(* CODESYS project CtaVisApps_1.0.0.0.library
   DocFormat: reStructuredText
   DefaultNamespace: CtaVisApps
   Version: 1.0.0.0
   Placeholder: CtaVisApps
   Company: CTA
   Description: Visu Apps Library der CTA
   CompiledLibraryCompatibilityVersion: CODESYS V3.5 SP16 Patch 3
   LanguageModelAttribute: qualified-access-only
   Title: CtaVisApps
   Author: SIS

Project tree, tasks and I/O mapping:
  libraries: CmpBitmapPool, 3.5.17.0 (System); Visu Utils, 4.5.0.0 (System); Standard, 3.5.18.0 (System); VisuElemBase, * (System); CtaVisSymbols, 1.0.0.0 (CTA); TextListUtils, * (System); VisuSymbols, 4.5.0.0 (System)
  40 Visualizations/
    APP/
      visualisation VIS_APP_BASE
      visualisation VIS_APP
    DESCTOP/
      visualisation VIS_DESCTOP_GVL
      visualisation VIS_DESCTOP_BASE
      visualisation VIS_DESCTOP_APP_LINE
      visualisation VIS_DESCTOP
  30 Program Organization Units/
    APP/
      function block FB_APP [ST]: DIALOG_NAME, ITF_BIG_SYBIL, ITF_LOW_SYBIL, ITF_PARENT, TEXTLIST, TEXTLISTID, PRESS_EVENT, ITF_CHILD, FB_INIT, ITF_SELF, ENABLED, DATA, DATA_SIZE, RELOAD_REQUEST, APP_NAME, ITF_DESCTOP
    DESCTOP/
      function block FB_DESCTOP [ST]: GET_APP, FIRST_APP, RETURN_APP, PATH, DialogClosed, LOWEST_CHILD, HOME, RELOAD_REQUEST
  00000000-0000-0000-0000-000000000000|D:\CoDeSys\LibrariesV3\trunk\Intern\CAA\CAA Template\3.4.0.0 draft\Placeholder.xml
  00000000-0000-0000-0000-000000000000|D:\CoDeSys\LibrariesV3\trunk\Intern\CAA\CAA Template\3.2.0.3 draft\Prefix.pdf
  00000000-0000-0000-0000-000000000000|D:\CoDeSys\LibrariesV3\trunk\Intern\CAA\CAA Template\3.5.2.0 draft\Placeholder.xml
  20 Structs/
  50 Images/
  10 Documenation/
    global variables VersionHistory
    global variables readMe
  21 Interface/
    interface ITF_APP: DIALOG_NAME, ITF_BIG_SYBIL, TEXTLISTID, ITF_LOW_SYBIL, TEXTLIST, PRESS_EVENT, ITF_CHILD, ITF_PARENT, ITF_SELF, ENABLED, DATA, DATA_SIZE, RELOAD_REQUEST, APP_NAME, ITF_DESCTOP
    interface ITF_DESCTOP: FIRST_APP, GET_APP, RETURN_APP, PATH, LOWEST_CHILD, HOME, RELOAD_REQUEST
  11 Library Parameter/
  12 Konstanten/
  60 Textlisten/
  13 Globale Variablen/
    global variables GVL_VISU_APPS
  5ce3da45-db07-42e7-a21c-a00fff4ed8f6|Icons\alert.svg
  5ce3da45-db07-42e7-a21c-a00fff4ed8f6|Icons\arrow-down.svg
  5ce3da45-db07-42e7-a21c-a00fff4ed8f6|Icons\arrow-down_square.svg
  5ce3da45-db07-42e7-a21c-a00fff4ed8f6|Icons\arrow-left_solo_black.svg
  5ce3da45-db07-42e7-a21c-a00fff4ed8f6|Icons\arrow-right_solo_black.svg
  5ce3da45-db07-42e7-a21c-a00fff4ed8f6|Icons\arrow-up.svg
  5ce3da45-db07-42e7-a21c-a00fff4ed8f6|Icons\calendar-range.svg
  5ce3da45-db07-42e7-a21c-a00fff4ed8f6|Icons\check.svg
  5ce3da45-db07-42e7-a21c-a00fff4ed8f6|Icons\clock-outline.svg
  5ce3da45-db07-42e7-a21c-a00fff4ed8f6|Icons\close_solo_black.svg
  5ce3da45-db07-42e7-a21c-a00fff4ed8f6|Icons\CtaInfo.svg
  5ce3da45-db07-42e7-a21c-a00fff4ed8f6|Icons\database_black.svg
  5ce3da45-db07-42e7-a21c-a00fff4ed8f6|Icons\delete_solo_black.svg
  5ce3da45-db07-42e7-a21c-a00fff4ed8f6|Icons\engine.svg
  5ce3da45-db07-42e7-a21c-a00fff4ed8f6|Icons\front_hand_Black.svg
  5ce3da45-db07-42e7-a21c-a00fff4ed8f6|Icons\front_hand_Yellow_Off.svg
  5ce3da45-db07-42e7-a21c-a00fff4ed8f6|Icons\gear.svg
  5ce3da45-db07-42e7-a21c-a00fff4ed8f6|Icons\home.svg
  5ce3da45-db07-42e7-a21c-a00fff4ed8f6|Icons\information-variant.svg
  5ce3da45-db07-42e7-a21c-a00fff4ed8f6|Icons\lightning-bolt-circle.svg
  5ce3da45-db07-42e7-a21c-a00fff4ed8f6|Icons\message.svg
  5ce3da45-db07-42e7-a21c-a00fff4ed8f6|Icons\message-alert-variant.svg
  5ce3da45-db07-42e7-a21c-a00fff4ed8f6|Icons\minus_solo_black.svg
  5ce3da45-db07-42e7-a21c-a00fff4ed8f6|Icons\plus_solo_black.svg
  5ce3da45-db07-42e7-a21c-a00fff4ed8f6|Icons\power_solo_black.svg
  5ce3da45-db07-42e7-a21c-a00fff4ed8f6|Icons\refresh_solo_black.svg
  5ce3da45-db07-42e7-a21c-a00fff4ed8f6|Icons\SearchFilter.svg
  5ce3da45-db07-42e7-a21c-a00fff4ed8f6|Icons\signal-celular-alt.svg
  5ce3da45-db07-42e7-a21c-a00fff4ed8f6|Icons\toggle-switch.svg
  5ce3da45-db07-42e7-a21c-a00fff4ed8f6|Icons\Modbus_Organization_Logo.svg
  5ce3da45-db07-42e7-a21c-a00fff4ed8f6|Icons\CheckboxUnchecked_withe.svg
  5ce3da45-db07-42e7-a21c-a00fff4ed8f6|Icons\lock_open_black.svg
  5ce3da45-db07-42e7-a21c-a00fff4ed8f6|Icons\check_green.svg
  5ce3da45-db07-42e7-a21c-a00fff4ed8f6|Icons\filter_black.svg
  5ce3da45-db07-42e7-a21c-a00fff4ed8f6|Icons\CtaLogo.png
  5ce3da45-db07-42e7-a21c-a00fff4ed8f6|Icons\Grafana_Logo.svg
  5ce3da45-db07-42e7-a21c-a00fff4ed8f6|Icons\hourglass_top.svg
  text list GlobalTextList
*)

// 10 Documenation/VersionHistory
(* 

.. image:: ../../Images/CTA_Logo.jpg
   :align: right
   :width: 15% 

**History**   


============ =========== =========== ============================================
**Date**     **Version** **Author**  **Change**
------------ ----------- ----------- --------------------------------------------
04.09.2023   0.0.0.1     SIS         Entwicklung Apps

============ =========== =========== ============================================


*)
VAR_GLOBAL
    stInfo : STRING:= '0.0.0.0, Vorlage, CTA';
END_VAR

// 10 Documenation/readMe
(*

**ReadMe**
 
|	**Empfehlung**
|
|	Mithilfe der CtaVisApps Library kann ein App Desctop erstellt werden mit minimalem Aufwand. Dazu muss die Visualisierung VIS_DESCTOP im Projekt implementiert werden.
|     
| *Beispiel*
+-----------------------+---------------------------------------------------------------------------------------------------------------------------------------------------------------------------------------------------------------------------------------------------------------------------------------------------------------------------------------------------------------------------------------------------------------------------------------+
| Beschreibung          |  Code                                                                                                                                                                                                                                                                                                                                                                                                                                 |
+=======================+=======================================================================================================================================================================================================================================================================================================================================================================================================================================+
| Deklaration           | .. code-block:: codesys                                                                                                                                                                                                                                                                                                                                                                                                               |
|                       |                                                                                                                                                                                                                                                            																																											|
|                       | 		APP_PFC200									:	CtaVisApps.FB_APP(0				,0)					:= 			(_ENABLED := TRUE,    _TEXTLIST	:= 'APPS',		_TEXTLISTID		:= 'PFC200',		_DIALOG_NAME	:= 'DIA_WBM');                       																																							            |
|                       |		APP_Management								:	CtaVisApps.FB_APP(0				,APP_PFC200)		:= 			(_ENABLED := TRUE,    _TEXTLIST	:= 'APPS',		_TEXTLISTID		:= 'MANAGEMENT',	_DIALOG_NAME	:= 'DIA_AnlagenManagement');     																																										 	|
|                       |   	APP_STVDA									: 	CtaVisApps.FB_APP(0				,APP_Management)	:= 			(_ENABLED := TRUE,    _TEXTLIST	:= 'APPS',		_TEXTLISTID		:= 'STVDA',			_DIALOG_NAME	:= ''	);                       																																									      	|
|						|			APP_F100								:	CtaVisApps.FB_APP(APP_STVDA		,0)					:= 			(_ENABLED := TRUE,    _TEXTLIST	:= 'APPS',		_TEXTLISTID		:= 'F100',			_DIALOG_NAME	:= ''	);                       																																							            	|
|						|				APP_F100S1							:	CtaVisApps.FB_APP(APP_F100		,0)					:= 			(_ENABLED := TRUE,    _TEXTLIST	:= 'APPS',		_TEXTLISTID		:= 'F100S1',		_DIALOG_NAME	:= ''	);                       																																									      	|
|                       | 					APP_100B011						:	CtaVisApps.FB_APP(APP_F100S1	,0)					:= 			(_ENABLED := TRUE,    _TEXTLIST	:= 'APPS',		_TEXTLISTID		:= '100B011',		_DIALOG_NAME	:= ''	);                       																																										 	|
| 						|					APP_100B012						:	CtaVisApps.FB_APP(APP_F100S1	,APP_100B011)		:= 			(_ENABLED := TRUE,    _TEXTLIST	:= 'APPS',		_TEXTLISTID		:= '100B012',		_DIALOG_NAME	:= ''	);                       																																											|
| 						|				APP_F100S2							:	CtaVisApps.FB_APP(APP_F100		,APP_F100S1)		:= 			(_ENABLED := TRUE,    _TEXTLIST	:= 'APPS',		_TEXTLISTID		:= 'F100S2',		_DIALOG_NAME	:= ''	);                       																																											|
| 						|					APP_100M021						:	CtaVisApps.FB_APP(APP_F100S2	,0)					:= 			(_ENABLED := TRUE,    _TEXTLIST	:= 'APPS',		_TEXTLISTID		:= '100M021',		_DIALOG_NAME	:= ''	);                       																																											|
| 						|				APP_F100S3							:	CtaVisApps.FB_APP(APP_F100		,APP_F100S2)		:= 			(_ENABLED := TRUE,    _TEXTLIST	:= 'APPS',		_TEXTLISTID		:= 'F100S3',		_DIALOG_NAME	:= ''	);                       																																											|
| 						|					APP_100M031						:	CtaVisApps.FB_APP(APP_F100S3	,0)					:= 			(_ENABLED := TRUE,    _TEXTLIST	:= 'APPS',		_TEXTLISTID		:= '100M031',		_DIALOG_NAME	:= ''	);                       																																											|
| 						|					APP_100M032						:	CtaVisApps.FB_APP(APP_F100S3	,APP_100M031)		:= 			(_ENABLED := TRUE,    _TEXTLIST	:= 'APPS',		_TEXTLISTID		:= '100M032',		_DIALOG_NAME	:= ''	);                       																																											|
| 						| 				APP_F100S4							:	CtaVisApps.FB_APP(APP_F100		,APP_F100S3)		:= 			(_ENABLED := TRUE,    _TEXTLIST	:= 'APPS',		_TEXTLISTID		:= 'F100S4',		_DIALOG_NAME	:= ''	);                       																																											|
| 						|					APP_100M041						:	CtaVisApps.FB_APP(APP_F100S4	,0)					:= 			(_ENABLED := TRUE,    _TEXTLIST	:= 'APPS',		_TEXTLISTID		:= '100M041',		_DIALOG_NAME	:= ''	);                       																																											|
| 						|					APP_100M042						:	CtaVisApps.FB_APP(APP_F100S4	,APP_100M041)		:= 			(_ENABLED := TRUE,    _TEXTLIST	:= 'APPS',		_TEXTLISTID		:= '100M042',		_DIALOG_NAME	:= ''	);                       																																											|
| 						|				APP_F100S5							:	CtaVisApps.FB_APP(APP_F100		,APP_F100S4)		:= 			(_ENABLED := TRUE,    _TEXTLIST	:= 'APPS',		_TEXTLISTID		:= 'F100S5',		_DIALOG_NAME	:= ''	);                       																																											|
| 						|					APP_100M051						:	CtaVisApps.FB_APP(APP_F100S5	,0)					:= 			(_ENABLED := TRUE,    _TEXTLIST	:= 'APPS',		_TEXTLISTID		:= '100M051',		_DIALOG_NAME	:= ''	);                       																																											|
| 						|					APP_100M052						:	CtaVisApps.FB_APP(APP_F100S5	,APP_100M051)		:= 			(_ENABLED := TRUE,    _TEXTLIST	:= 'APPS',		_TEXTLISTID		:= '100M052',		_DIALOG_NAME	:= ''	);                       																																											|
| 						|				APP_F100S6							:	CtaVisApps.FB_APP(APP_F100		,APP_F100S5)		:= 			(_ENABLED := TRUE,    _TEXTLIST	:= 'APPS',		_TEXTLISTID		:= 'F100S6',		_DIALOG_NAME	:= ''	);                       																																											|
| 						|					APP_100M061						:	CtaVisApps.FB_APP(APP_F100S6	,0)					:= 			(_ENABLED := TRUE,    _TEXTLIST	:= 'APPS',		_TEXTLISTID		:= '100M061',		_DIALOG_NAME	:= ''	);                       																																											|
| 						|					APP_100M062						:	CtaVisApps.FB_APP(APP_F100S6	,APP_100M061)		:= 			(_ENABLED := TRUE,    _TEXTLIST	:= 'APPS',		_TEXTLISTID		:= '100M062',		_DIALOG_NAME	:= ''	);                       																																											|
| 						|				APP_F100S7							:	CtaVisApps.FB_APP(APP_F100		,APP_F100S6)		:= 			(_ENABLED := TRUE,    _TEXTLIST	:= 'APPS',		_TEXTLISTID		:= 'F100S7',		_DIALOG_NAME	:= ''	);                       																																											|
| 						|					APP_100M071						:	CtaVisApps.FB_APP(APP_F100S7	,0)					:= 			(_ENABLED := TRUE,    _TEXTLIST	:= 'APPS',		_TEXTLISTID		:= '100M071',		_DIALOG_NAME	:= ''	);                       																																											|
| 						|					APP_100M072						:	CtaVisApps.FB_APP(APP_F100S7	,APP_100M071)		:= 			(_ENABLED := TRUE,    _TEXTLIST	:= 'APPS',		_TEXTLISTID		:= '100M072',		_DIALOG_NAME	:= ''	);                       																																											|
| 						|				APP_F100S8							:	CtaVisApps.FB_APP(APP_F100		,APP_F100S7)		:= 			(_ENABLED := TRUE,    _TEXTLIST	:= 'APPS',		_TEXTLISTID		:= 'F100S8',		_DIALOG_NAME	:= ''	);                       																																											|
| 						|					APP_100B081						:	CtaVisApps.FB_APP(APP_F100S8	,0)					:= 			(_ENABLED := TRUE,    _TEXTLIST	:= 'APPS',		_TEXTLISTID		:= '100B081',		_DIALOG_NAME	:= ''	);                       																																											|
| 						|					APP_100B082						:	CtaVisApps.FB_APP(APP_F100S8	,APP_100B081)		:= 			(_ENABLED := TRUE,    _TEXTLIST	:= 'APPS',		_TEXTLISTID		:= '100B082',		_DIALOG_NAME	:= ''	);                       																																											|
| 						|				APP_F100S9							:	CtaVisApps.FB_APP(APP_F100		,APP_F100S8)		:= 			(_ENABLED := TRUE,    _TEXTLIST	:= 'APPS',		_TEXTLISTID		:= 'F100S9',		_DIALOG_NAME	:= ''	);                       																																											|
| 						|					APP_100B091						:	CtaVisApps.FB_APP(APP_F100S9	,0)					:= 			(_ENABLED := TRUE,    _TEXTLIST	:= 'APPS',		_TEXTLISTID		:= '100B091',		_DIALOG_NAME	:= ''	);                       																																											|
| 						|					APP_100B092						:	CtaVisApps.FB_APP(APP_F100S9	,APP_100B091)		:= 			(_ENABLED := TRUE,    _TEXTLIST	:= 'APPS',		_TEXTLISTID		:= '100B092',		_DIALOG_NAME	:= ''	);                       																																											|
| 						|				APP_F100S10							:	CtaVisApps.FB_APP(APP_F100		,APP_F100S9)		:= 			(_ENABLED := TRUE,    _TEXTLIST	:= 'APPS',		_TEXTLISTID		:= 'F100S10',		_DIALOG_NAME	:= ''	);                       																																											|
| 						|					APP_100M101						:	CtaVisApps.FB_APP(APP_F100S10	,0)					:= 			(_ENABLED := TRUE,    _TEXTLIST	:= 'APPS',		_TEXTLISTID		:= '100M101',		_DIALOG_NAME	:= ''	);                       																																											|
| 						|				APP_F100S11							:	CtaVisApps.FB_APP(APP_F100		,APP_F100S10)		:= 			(_ENABLED := TRUE,    _TEXTLIST	:= 'APPS',		_TEXTLISTID		:= 'F100S11',		_DIALOG_NAME	:= ''	);	                     																																											|
| 						|					APP_100E111						:	CtaVisApps.FB_APP(APP_F100S11	,0)					:= 			(_ENABLED := TRUE,    _TEXTLIST	:= 'APPS',		_TEXTLISTID		:= '100E111',		_DIALOG_NAME	:= ''	);                       																																											|
| 						|					APP_100E112						:	CtaVisApps.FB_APP(APP_F100S11	,APP_100E111)		:= 			(_ENABLED := TRUE,    _TEXTLIST	:= 'APPS',		_TEXTLISTID		:= '100E112',		_DIALOG_NAME	:= ''	);                      																																											|
| 						|			APP_F200								:	CtaVisApps.FB_APP(APP_STVDA		,APP_F100)			:= 			(_ENABLED := TRUE,    _TEXTLIST	:= 'APPS',		_TEXTLISTID		:= 'F200',			_DIALOG_NAME	:= ''	);                       																																											|
| 						|	                                                                                                                                                                                             																																																										|
| 						|																												                                                                                                                                                                                                                                                                                                                    	|
+-----------------------+---------------------------------------------------------------------------------------------------------------------------------------------------------------------------------------------------------------------------------------------------------------------------------------------------------------------------------------------------------------------------------------------------------------------------------------+
| Code					| .. code-block:: codesys 															                                                                                                                                                                                                                                                                                                                    								|
| 						|																												                                                                                                                                                                                                                                                                                                                    	|
| 						|	GVL_VISU_APP.DESCTOP();																																																																																																				|
| 						|	GVL_VISU_APP.DESCTOP.FIRST_APP(APP_PFC200);																											                                                                                                                                                                                                                                                                                |
| 						|																												                                                                                                                                                                                                                                                                                                                    	|
+-----------------------+---------------------------------------------------------------------------------------------------------------------------------------------------------------------------------------------------------------------------------------------------------------------------------------------------------------------------------------------------------------------------------------------------------------------------------------+
*)

VAR_GLOBAL
    xReadMeDone              :   BOOL;
END_VAR

// 13 Globale Variablen/GVL_VISU_APPS
{attribute 'qualified_only'}
{attribute 'linkalways'}
VAR_GLOBAL
	DESCTOP										: FB_DESCTOP;
END_VAR

// 21 Interface/ITF_APP
INTERFACE ITF_APP EXTENDS __System.Iqueryinterface

PROPERTY DIALOG_NAME : STRING
GET
END_GET
END_PROPERTY

PROPERTY ITF_BIG_SYBIL : ITF_APP
SET
END_SET
GET
END_GET
END_PROPERTY

PROPERTY TEXTLISTID : STRING
GET
END_GET
END_PROPERTY

PROPERTY ITF_LOW_SYBIL : ITF_APP
SET
END_SET
GET
END_GET
END_PROPERTY

PROPERTY TEXTLIST : STRING
GET
END_GET
END_PROPERTY

PROPERTY PRESS_EVENT : BOOL
SET
END_SET
GET
END_GET
END_PROPERTY

PROPERTY ITF_CHILD : ITF_APP
SET
END_SET
GET
END_GET
END_PROPERTY

PROPERTY ITF_PARENT : ITF_APP
GET
END_GET
SET
END_SET
END_PROPERTY

PROPERTY ITF_SELF : ITF_APP
GET
END_GET
END_PROPERTY

PROPERTY ENABLED : BOOL
SET
END_SET
GET
END_GET
END_PROPERTY

PROPERTY DATA : POINTER TO BYTE
GET
END_GET
END_PROPERTY

PROPERTY DATA_SIZE : UDINT
GET
END_GET
END_PROPERTY

PROPERTY RELOAD_REQUEST : BOOL
SET
END_SET
GET
END_GET
END_PROPERTY

PROPERTY APP_NAME : STRING
GET
END_GET
END_PROPERTY

PROPERTY ITF_DESCTOP : ITF_DESCTOP
SET
END_SET
END_PROPERTY

END_INTERFACE

// 21 Interface/ITF_DESCTOP
INTERFACE ITF_DESCTOP EXTENDS __System.Iqueryinterface

METHOD FIRST_APP
VAR_INPUT
	ITF_APP	:	ITF_APP;
END_VAR
END_METHOD

METHOD GET_APP : ITF_APP
VAR_INPUT
	usiChildNr		:	USINT;
END_VAR
END_METHOD

METHOD RETURN_APP
VAR_INPUT
END_VAR
END_METHOD

PROPERTY PATH : STRING(255)
GET
END_GET
END_PROPERTY

PROPERTY LOWEST_CHILD : USINT
GET
END_GET
END_PROPERTY

METHOD HOME
VAR_INPUT
END_VAR
END_METHOD

METHOD RELOAD_REQUEST
VAR_INPUT
END_VAR
END_METHOD

END_INTERFACE

// 30 Program Organization Units/APP/FB_APP
FUNCTION_BLOCK FB_APP IMPLEMENTS ITF_APP
VAR_INPUT
	_TEXTLIST		:	STRING;							// Textlist with App Text 
	_TEXTLISTID		:	STRING(20);						// Textlist Id
	_DIALOG_NAME	:	STRING;							// Dialog Name to Oppen if needed
	_ENABLED		:	BOOL;							// Mark as Enabled tho show
	_DATA			:	POINTER TO BYTE;				// Data fore Dialog 
	_DATA_SIZE		:	UDINT;							// Size of Data
END_VAR
VAR_OUTPUT
END_VAR
VAR
	{attribute 'hide'}
	_PRESS_EVENT	:	BOOL;
	_RELOD_REQUEST	:	BOOL;
	{attribute 'hide'}
	_ITF_PARENT		:	ITF_APP;
	{attribute 'hide'}
	_ITF_BIG_SYBIL	:	ITF_APP;
	{attribute 'hide'}
	_ITF_LOW_SYBIL	:	ITF_APP;
	{attribute 'hide'}
	_ITF_CHILD		:	ITF_APP;
	{attribute 'hide'}
	_ITF_DESCTOP	:	ITF_DESCTOP;
END_VAR

PROPERTY DIALOG_NAME : STRING
GET
DIALOG_NAME := _DIALOG_NAME;
END_GET
END_PROPERTY

{attribute 'estimated-stack-usage' := '40'}
PROPERTY ITF_BIG_SYBIL : ITF_APP
GET
ITF_BIG_SYBIL := _ITF_BIG_SYBIL;
END_GET
SET
_ITF_BIG_SYBIL := ITF_BIG_SYBIL;
IF __QUERYINTERFACE(_ITF_BIG_SYBIL,_ITF_BIG_SYBIL) THEN
	IF _ITF_BIG_SYBIL.ITF_LOW_SYBIL <> ITF_SELF THEN
		_ITF_BIG_SYBIL.ITF_LOW_SYBIL := THIS^;
	END_IF;
END_IF;
END_SET
END_PROPERTY

PROPERTY ITF_LOW_SYBIL : ITF_APP
GET
ITF_LOW_SYBIL := _ITF_LOW_SYBIL;
END_GET
SET
_ITF_LOW_SYBIL := ITF_LOW_SYBIL;
IF __QUERYINTERFACE(_ITF_LOW_SYBIL,_ITF_LOW_SYBIL) THEN
	IF _ITF_LOW_SYBIL.ITF_BIG_SYBIL <> ITF_SELF THEN
		_ITF_LOW_SYBIL.ITF_BIG_SYBIL := THIS^;
	END_IF;
END_IF;
END_SET
END_PROPERTY

{attribute 'estimated-stack-usage' := '40'}
PROPERTY ITF_PARENT : ITF_APP
GET
ITF_PARENT := _ITF_PARENT;
END_GET
SET
_ITF_PARENT := ITF_PARENT;
IF __QUERYINTERFACE(_ITF_PARENT,_ITF_PARENT) THEN
	IF _ITF_PARENT.ITF_CHILD <> ITF_SELF AND ITF_BIG_SYBIL = 0 THEN
		_ITF_PARENT.ITF_CHILD := THIS^;
	END_IF;
END_IF;
END_SET
END_PROPERTY

PROPERTY TEXTLIST : STRING
GET
TEXTLIST := _TEXTLIST;
END_GET
END_PROPERTY

PROPERTY TEXTLISTID : STRING
GET
TEXTLISTID := _TEXTLISTID;
END_GET
END_PROPERTY

PROPERTY PRESS_EVENT : BOOL
SET
_PRESS_EVENT := PRESS_EVENT;
IF _PRESS_EVENT THEN
	RELOAD_REQUEST := _PRESS_EVENT;
END_IF;
END_SET
GET
PRESS_EVENT := _PRESS_EVENT;
END_GET
END_PROPERTY

PROPERTY ITF_CHILD : ITF_APP
SET
_ITF_CHILD := ITF_CHILD;
IF __QUERYINTERFACE(_ITF_CHILD,_ITF_CHILD) THEN
	IF _ITF_CHILD.ITF_PARENT <> ITF_SELF THEN
		_ITF_CHILD.ITF_PARENT := THIS^;
	END_IF;
END_IF;
END_SET
GET
ITF_CHILD := _ITF_CHILD;
END_GET
END_PROPERTY

//FB_Init ist immer implizit verfügbar und wird primär für die Initialisierung verwendet.
//Der Rückgabewert wird nicht ausgewertet. Für gezielte Einflussnahme können Sie
//die Methoden explizit deklarieren und darin mit dem Standard-Initialisierungscode 
//zusätzlichen Code bereitstellen. Sie können den Rückgabewert auswerten.
METHOD FB_Init: BOOL
VAR_INPUT    
	bInitRetains: BOOL; // TRUE: Die Retain-Variablen werden initialisiert (Reset warm / Reset kalt)    
	bInCopyCode: BOOL;  // TRUE: Die Instanz wird danach in den Kopiercode kopiert (Online-Change)
	ITF_PARENT_INI		:	ITF_APP;
	ITF_BIG_SYBIL_INI	:	ITF_APP;
END_VAR
ITF_BIG_SYBIL 	:= ITF_BIG_SYBIL_INI;
ITF_PARENT 		:= ITF_PARENT_INI;
END_METHOD

PROPERTY ITF_SELF : ITF_APP
GET
ITF_SELF := THIS^;
END_GET
END_PROPERTY

PROPERTY ENABLED : BOOL
SET
_ENABLED := ENABLED;
END_SET
GET
ENABLED := _ENABLED;
END_GET
END_PROPERTY

PROPERTY DATA : POINTER TO BYTE
GET
DATA := _DATA;
END_GET
END_PROPERTY

PROPERTY DATA_SIZE : UDINT
GET
DATA_SIZE := _DATA_SIZE;
END_GET
END_PROPERTY

{attribute 'estimated-stack-usage' := '40'}
PROPERTY RELOAD_REQUEST : BOOL
SET
VAR
END_VAR
{attribute 'estimated-stack-usage' := '127'}
_RELOD_REQUEST := RELOAD_REQUEST;
(* Positive Event call Up *)
IF _RELOD_REQUEST THEN
	(* Check if Parent is valid *)
	IF __QUERYINTERFACE(_ITF_PARENT,_ITF_PARENT) THEN
		_ITF_PARENT.RELOAD_REQUEST := _RELOD_REQUEST;
	(* Elseif  inform Big Sybil *)
	ELSIF __QUERYINTERFACE(_ITF_BIG_SYBIL,_ITF_BIG_SYBIL) THEN
		_ITF_BIG_SYBIL.RELOAD_REQUEST := _RELOD_REQUEST;
	(* Elseif Call Desctop *)
	ELSIF __QUERYINTERFACE(_ITF_DESCTOP,_ITF_DESCTOP) THEN
		_ITF_DESCTOP.RELOAD_REQUEST();
	END_IF;
(* Negative Event call Down *)
ELSE
	(* Check if Child is valid & inform Child*)
	IF __QUERYINTERFACE(_ITF_CHILD,_ITF_CHILD) THEN
		_ITF_CHILD.RELOAD_REQUEST := _RELOD_REQUEST;
	END_IF;
	(* Check if Child is valid & inform Child*)
	IF __QUERYINTERFACE(_ITF_LOW_SYBIL,_ITF_LOW_SYBIL) THEN
		_ITF_LOW_SYBIL.RELOAD_REQUEST := _RELOD_REQUEST;
	END_IF;	
END_IF;
END_SET
GET
RELOAD_REQUEST := _RELOD_REQUEST;
END_GET
END_PROPERTY

PROPERTY APP_NAME : STRING
GET
__TRY
	TLU.GetText(_TEXTLIST,_TEXTLISTID,ADR(APP_NAME),SIZEOF(APP_NAME));
__CATCH
APP_NAME := '';
__ENDTRY
END_GET
END_PROPERTY

PROPERTY ITF_DESCTOP : ITF_DESCTOP
SET
_ITF_DESCTOP := ITF_DESCTOP;
END_SET
END_PROPERTY

END_FUNCTION_BLOCK

// 30 Program Organization Units/DESCTOP/FB_DESCTOP
{attribute 'hide'}
FUNCTION_BLOCK FB_DESCTOP IMPLEMENTS ITF_DESCTOP , VisuElems.IDialogCloseListener
VAR_INPUT
END_VAR
VAR_OUTPUT
END_VAR
VAR
	_FIRST_APP			:	ITF_APP;
	
	_RETURN_APP			:	ITF_APP;
	
	_AY_APP				:	ARRAY[0..39] OF ITF_APP;
	
	diFor				:	DINT;
	diFor2				:	DINT;
	xInitDone			:	BOOL;
	fbOpenDialog 		: 	VU.FbOpenDialogExtended;
	FbCloseDialog		:	VU.FbCloseDialog;
	usiLowestChild		:	USINT;
	usiLowestChildTemp	:	USINT;
END_VAR

METHOD GET_APP : ITF_APP
VAR_INPUT
	usiChildNr		:	USINT;
END_VAR
(* Check if Request is lower then lowest Child *)
IF usiChildNr <= usiLowestChild THEN
	(* Check Array Bounds *)
	IF TO_DINT(usiChildNr) >= LOWER_BOUND(_AY_APP,1) AND TO_DINT(usiChildNr) <= UPPER_BOUND(_AY_APP,1) THEN 
		(* Gett App *)
		GET_APP := _AY_APP[usiChildNr];
	ELSE
		GET_APP := 0;
	END_IF;
ELSE
	GET_APP :=  0;
END_IF;
END_METHOD

METHOD FIRST_APP
VAR_INPUT
	ITF_APP	:	ITF_APP;
END_VAR
VAR
	diForTemp	:	DINT;
END_VAR
(* Check if First App is diffrent *)
IF ITF_APP <> _FIRST_APP THEN
	_FIRST_APP := ITF_APP;
	IF __QUERYINTERFACE(_FIRST_APP,_FIRST_APP) THEN
		_FIRST_APP.ITF_DESCTOP := THIS^;
	END_IF
	xInitDone := FALSE;
END_IF;
(* Init Array *)
IF NOT xInitDone THEN
	(* Check if valid First App *)
	IF __QUERYINTERFACE(_FIRST_APP,_FIRST_APP) THEN
		_FIRST_APP.RELOAD_REQUEST := TRUE;
		_AY_APP[0] := _FIRST_APP;
	END_IF;
	FOR diForTemp := LOWER_BOUND(_AY_APP,1) TO UPPER_BOUND(_AY_APP,1)-1 DO
		(* Check if valid *)
		IF __QUERYINTERFACE(_AY_APP[diForTemp],_AY_APP[diForTemp]) THEN
			(* Add Low Sybil *)
			_AY_APP[diForTemp + 1]	:= _AY_APP[diForTemp].ITF_LOW_SYBIL;
			(* Check if valid Low Sybil *)
			IF __QUERYINTERFACE(_AY_APP[diForTemp + 1],_AY_APP[diForTemp + 1]) THEN
				(* Add Big Sybil to Low Sybil *)
				_AY_APP[diForTemp + 1].ITF_BIG_SYBIL := _AY_APP[diForTemp];
			ELSE
				EXIT;
			END_IF;
		END_IF;
	END_FOR
	(* Init Done *)
	xInitDone := TRUE;
	RELOAD_REQUEST();
END_IF;
END_METHOD

METHOD RETURN_APP
VAR_INPUT
END_VAR
VAR
	ITF_TEMP_BIG_SYBIL	:	ITF_APP;
	ITF_BIGEST_SYBIL	:	ITF_APP;
	diForTemp			:	DINT;
END_VAR
(* Check if Retund App is Valid *)
IF __QUERYINTERFACE(_RETURN_APP,_RETURN_APP) THEN
	(* Get Big Sybil of Return App *)
	ITF_TEMP_BIG_SYBIL := _RETURN_APP.ITF_BIG_SYBIL;
	ITF_BIGEST_SYBIL   := _RETURN_APP;
	(* Repeat get big Sybil until the Bigest is found *)
	REPEAT 
		(* Check if valid *)
		IF __QUERYINTERFACE(ITF_TEMP_BIG_SYBIL,ITF_TEMP_BIG_SYBIL) THEN
			(* Get the new Bigest Sybil *)
			ITF_BIGEST_SYBIL	:= ITF_TEMP_BIG_SYBIL;
			ITF_TEMP_BIG_SYBIL := ITF_TEMP_BIG_SYBIL.ITF_BIG_SYBIL;	
		ELSE
			ITF_TEMP_BIG_SYBIL := 0;
		END_IF;
	UNTIL ITF_TEMP_BIG_SYBIL = 0
	END_REPEAT
	(* Set the Biggest Sybil as App Start point *)
	_AY_APP[0] :=  ITF_BIGEST_SYBIL;
	(* Set the new Return App with the Parent of the Biggest Sybil *)
	_RETURN_APP := ITF_BIGEST_SYBIL.ITF_PARENT;
	(* Load the requieret Apps *)
	FOR diForTemp := LOWER_BOUND(_AY_APP,1) TO UPPER_BOUND(_AY_APP,1)-1 DO
		(* Clean App *)
		_AY_APP[diForTemp + 1]	:= 0;
		(* Check if Valid *)
		IF __QUERYINTERFACE(_AY_APP[diForTemp],_AY_APP[diForTemp]) THEN
			(* Set Low Sybil *)
			_AY_APP[diForTemp + 1]	:= _AY_APP[diForTemp].ITF_LOW_SYBIL;
			(* Check if Low Sybil is valid *)
			IF __QUERYINTERFACE(_AY_APP[diForTemp + 1],_AY_APP[diForTemp + 1]) THEN
				(* Set Big Sybil *)
				_AY_APP[diForTemp + 1].ITF_BIG_SYBIL := _AY_APP[diForTemp];
			END_IF;
		END_IF;
	END_FOR;	
	_AY_APP[0].RELOAD_REQUEST := TRUE;
ELSE
	xInitDone := FALSE;
END_IF;
END_METHOD

PROPERTY PATH : STRING(255)
GET
VAR
	ITF_TEMP_PARENT	:	ITF_APP;
	stTemp			:	STRING;
	stTextListTemp	:	STRING;
	stTextListIdTemp:	STRING;
END_VAR
PATH := '/';
IF __QUERYINTERFACE(_RETURN_APP,_RETURN_APP) THEN
	ITF_TEMP_PARENT := _RETURN_APP.ITF_PARENT;	
	__TRY
		stTextListTemp 		:= _RETURN_APP.TEXTLIST;
		stTextListIdTemp 	:=_RETURN_APP.TEXTLISTID;
		TLU.GetText(stTextListTemp,stTextListIdTemp,ADR(stTemp),SIZEOF(stTemp));
	__CATCH
		stTemp := '';
	__ENDTRY
	PATH := stTemp;
	REPEAT
		IF __QUERYINTERFACE(ITF_TEMP_PARENT,ITF_TEMP_PARENT) THEN
			__TRY
				stTemp := '';
				stTextListTemp 		:= ITF_TEMP_PARENT.TEXTLIST;
				stTextListIdTemp 	:= ITF_TEMP_PARENT.TEXTLISTID;
				TLU.GetText(stTextListTemp,stTextListIdTemp,ADR(stTemp),SIZEOF(stTemp));
			__CATCH
				stTemp := '';
			__ENDTRY
			PATH := CONCAT(stTemp,CONCAT(' / ',PATH));		
			ITF_TEMP_PARENT := ITF_TEMP_PARENT.ITF_PARENT;
		ELSE
			ITF_TEMP_PARENT := 0;
		END_IF
	UNTIL
		ITF_TEMP_PARENT = 0 
	END_REPEAT	
	PATH := CONCAT(' / ',PATH);		
END_IF;
END_GET
END_PROPERTY

(* Notification, that a dialog is closed.*)
METHOD DialogClosed
VAR_INPUT
	(* The IVisualisationDialog instance, that was closed*)
	itfDialog	: VisuElems.IVisualisationDialog;
	(* A pointer to the client data*)
	pClientData	: POINTER TO VisuElems.VisuStructClientData;
END_VAR
	FbCloseDialog(itfClientFilter 	:= VU.Globals.AllClients,
				  xExecute			:= FALSE,
				  sDialogName 		:= itfDialog.GetName(TRUE));
				  
	FbCloseDialog(itfClientFilter 	:= VU.Globals.AllClients,
				  xExecute			:= TRUE,
				  sDialogName 		:= itfDialog.GetName(TRUE));
END_METHOD

PROPERTY LOWEST_CHILD : USINT
GET
LOWEST_CHILD := usiLowestChild;
END_GET
END_PROPERTY

METHOD HOME
VAR_INPUT
END_VAR
VAR
	diForTemp	:	DINT;
END_VAR
(* Check if valid First App *)
IF __QUERYINTERFACE(_FIRST_APP,_FIRST_APP) THEN
	_FIRST_APP.RELOAD_REQUEST := TRUE;
	_RETURN_APP	:= _FIRST_APP.ITF_PARENT;
	_AY_APP[0] := _FIRST_APP;
END_IF;
FOR diForTemp := LOWER_BOUND(_AY_APP,1) TO UPPER_BOUND(_AY_APP,1)-1 DO
	(* Clean Table row *)
	_AY_APP[diForTemp + 1]	:= 0;
	(* Check if valid *)
	IF __QUERYINTERFACE(_AY_APP[diForTemp],_AY_APP[diForTemp]) THEN
		(* Add Low Sybil *)
		_AY_APP[diForTemp + 1]	:= _AY_APP[diForTemp].ITF_LOW_SYBIL;
		(* Check if valid Low Sybil *)
		IF __QUERYINTERFACE(_AY_APP[diForTemp + 1],_AY_APP[diForTemp + 1]) THEN
			(* Add Big Sybil to Low Sybil *)
			_AY_APP[diForTemp + 1].ITF_BIG_SYBIL := _AY_APP[diForTemp];
		END_IF;
	END_IF;
END_FOR
END_METHOD

METHOD RELOAD_REQUEST
VAR_INPUT
END_VAR
(* Check if Init Done *)
IF xInitDone THEN
	IF _FIRST_APP.RELOAD_REQUEST THEN
		(* Repeat fore all *)
		FOR diFor := LOWER_BOUND(_AY_APP,1) TO UPPER_BOUND(_AY_APP,1)-1 DO
			(* Check if valid *)
			IF __QUERYINTERFACE(_AY_APP[diFor],_AY_APP[diFor]) THEN
				(* Count Childs *)
				usiLowestChildTemp := TO_USINT(diFor + 1);
				(*Check witch has the Press event *)
				IF _AY_APP[diFor].PRESS_EVENT THEN
					(* Set to False *)
					_AY_APP[diFor].PRESS_EVENT := FALSE;
					(* Check if Dialog should be oppened or go down *)
					IF _AY_APP[diFor].DIALOG_NAME = '' THEN
						(* Set new Return App *)
						_RETURN_APP := _AY_APP[diFor];
						(* Set new start app *)
						_AY_APP[0] :=  _AY_APP[diFor].ITF_CHILD;
						(* Reload Table *)
						FOR diFor2 := LOWER_BOUND(_AY_APP,1) TO UPPER_BOUND(_AY_APP,1)-1 DO
							(* Clean Table row *)
							_AY_APP[diFor2 + 1]	:= 0;
							(* Check if valid *)
							IF __QUERYINTERFACE(_AY_APP[diFor2],_AY_APP[diFor2]) THEN
								(* Set the Parent *)
								_AY_APP[diFor2].ITF_PARENT := _RETURN_APP;
								(* Set Reload *)
								_AY_APP[diFor2].RELOAD_REQUEST := TRUE;
								(* Set Low Sybil *)
								_AY_APP[diFor2 + 1]	:= _AY_APP[diFor2].ITF_LOW_SYBIL;
								(* Check if Low Sybil is valid *)
								IF __QUERYINTERFACE(_AY_APP[diFor2 + 1],_AY_APP[diFor2 + 1]) THEN
									_AY_APP[diFor2 + 1].ITF_BIG_SYBIL := _AY_APP[diFor2];
								END_IF;
							END_IF;
						END_FOR;
					ELSE
						(* Close Dialog *)
						fbOpenDialog(	sDialogName 				:= _AY_APP[diFor].DIALOG_NAME,
										xModal 						:= FALSE, 
										pTopLeftPosition 			:= 0, 
										itfClientFilter 			:= VU.Globals.CurrentClient,
										xExecute	 				:= FALSE, 
										pbyDialogInterfaceData 		:= _AY_APP[diFor].DATA,
										udiDialogInterfaceDataSize 	:= _AY_APP[diFor].DATA_SIZE, 
										itfDialogCloseListener 		:= THIS^,
										pbyTagForDialogClosed		:= _AY_APP[diFor].DATA);
						(* Open Dialog *)			
						fbOpenDialog(	sDialogName 				:= _AY_APP[diFor].DIALOG_NAME,
										xModal 						:= FALSE, 
										pTopLeftPosition 			:= 0, 
										itfClientFilter 			:= VU.Globals.CurrentClient,
										xExecute	 				:= TRUE, 
										pbyDialogInterfaceData 		:= _AY_APP[diFor].DATA,
										udiDialogInterfaceDataSize 	:= _AY_APP[diFor].DATA_SIZE, 
										itfDialogCloseListener 		:= THIS^,
										pbyTagForDialogClosed		:= _AY_APP[diFor].DATA); 	
					END_IF;		
				END_IF;
			END_IF;
		END_FOR
		(* Set Count Child *)
		usiLowestChild := usiLowestChildTemp;
		(* Rload Request Done *)
		_FIRST_APP.RELOAD_REQUEST := FALSE;
	END_IF;
END_IF;
END_METHOD

END_FUNCTION_BLOCK

// 40 Visualizations/APP/VIS_APP_BASE
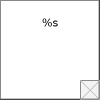
VISUALIZATION VIS_APP_BASE  // 100x100
VAR_INPUT
	ITF_APP_IN	:	ITF_APP;
END_VAR
    Textfield (2,15 96x65), "%s", text variable: ITF_APP_IN.APP_NAME
    RoundedRectangle (0,0 100x100)
        OnMouseClick: execute { ITF_APP_IN.PRESS_EVENT := TRUE; }
    Image (80,80 20x20), invisible if: ITF_APP_IN.ENABLED, image: CtaVisSymbols.ImagePool.close
    Image (80,80 20x20), invisible if: NOT ITF_APP_IN.ENABLED, image: CtaVisSymbols.ImagePool.check_green
END_VISUALIZATION

// 40 Visualizations/APP/VIS_APP
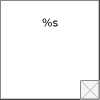
VISUALIZATION VIS_APP  // 100x100
VAR_INPUT
	ITF_APP_IN	:	ITF_APP;
END_VAR
    Frame (0,0 100x100), invisible if: NOT __Queryinterface(ITF_APP_IN,ITF_APP_IN)
        shows VIS_APP_BASE(ITF_APP_IN := ITF_APP_IN)
END_VISUALIZATION

// 40 Visualizations/DESCTOP/VIS_DESCTOP_GVL
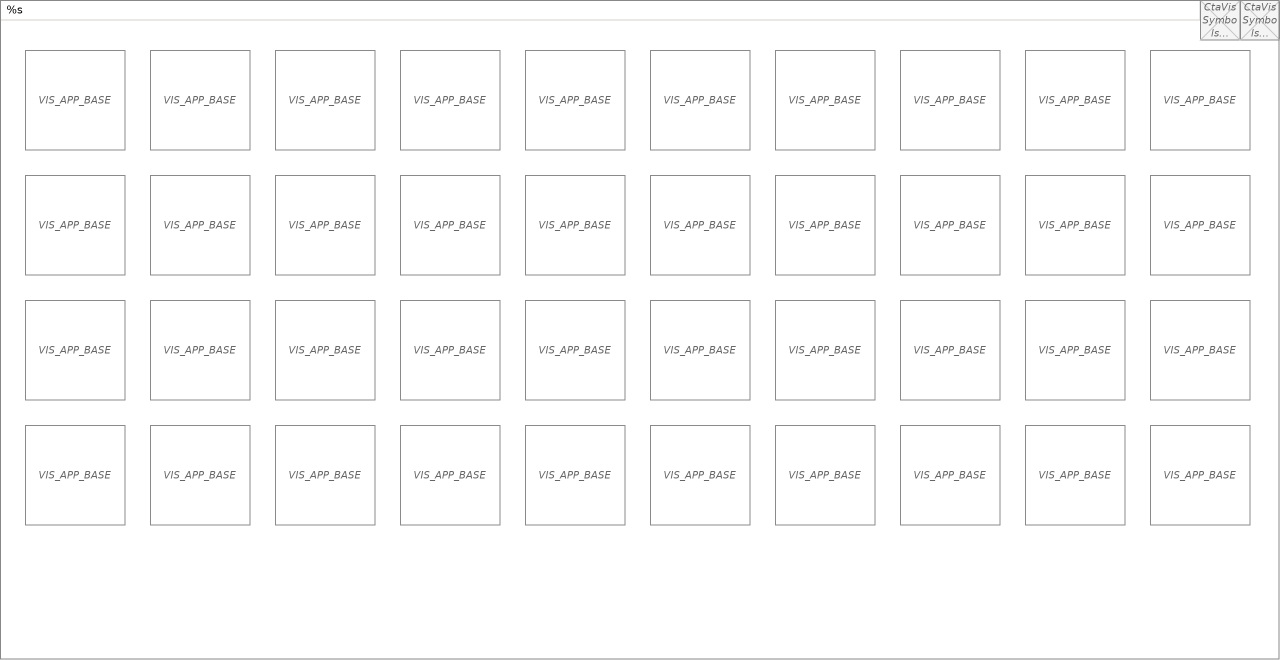
VISUALIZATION VIS_DESCTOP_GVL  // 1280x660
VAR_INPUT
	ITF_DESCTOP_IN : ITF_DESCTOP;
END_VAR
    Frame (0,0 1280x660), invisible if: NOT __Queryinterface(ITF_DESCTOP_IN,ITF_DESCTOP_IN)
        shows VIS_DESCTOP_BASE(ITF_DESCTOP_IN := ITF_DESCTOP_IN)
END_VISUALIZATION

// 40 Visualizations/DESCTOP/VIS_DESCTOP_BASE
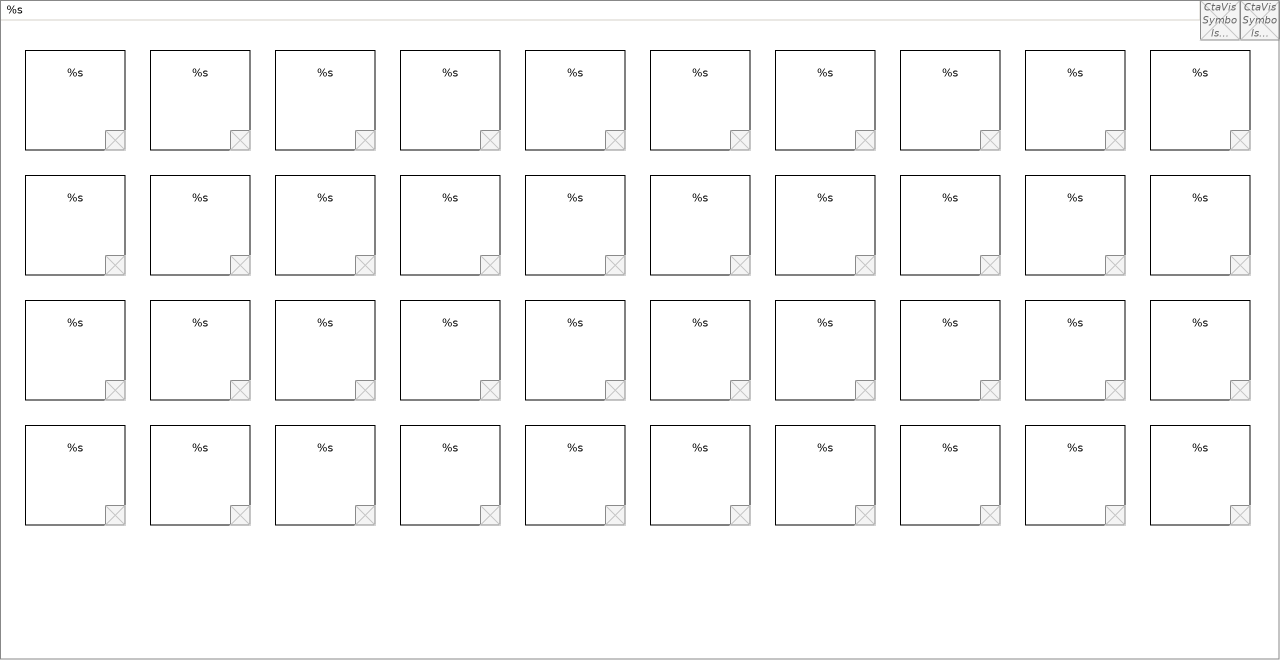
VISUALIZATION VIS_DESCTOP_BASE  // 1280x660
VAR_INPUT
	ITF_DESCTOP_IN : ITF_DESCTOP;
END_VAR
    Textfield (0,0 1200x20), "%s", text variable: ITF_DESCTOP_IN.PATH
    Image (1200,0 40x40), image: CtaVisSymbols.ImagePool.arrow-left_solo_black
        OnMouseClick: execute { ITF_DESCTOP_IN.RETURN_APP(); }
    Frame (0,50 1280x100), invisible if: ITF_DESCTOP_IN.LOWEST_CHILD = 0
        shows VIS_DESCTOP_APP_LINE(usiStartNr := 0, ITF_DESCTOP_IN := ITF_DESCTOP_IN)
    Frame (0,175 1280x100), invisible if: ITF_DESCTOP_IN.LOWEST_CHILD < 10
        shows VIS_DESCTOP_APP_LINE(usiStartNr := 10, ITF_DESCTOP_IN := ITF_DESCTOP_IN)
    Frame (0,300 1280x100), invisible if: ITF_DESCTOP_IN.LOWEST_CHILD < 20
        shows VIS_DESCTOP_APP_LINE(usiStartNr := 20, ITF_DESCTOP_IN := ITF_DESCTOP_IN)
    Frame (0,425 1280x100), invisible if: ITF_DESCTOP_IN.LOWEST_CHILD < 30
        shows VIS_DESCTOP_APP_LINE(usiStartNr := 30, ITF_DESCTOP_IN := ITF_DESCTOP_IN)
    Image (1240,0 40x40), image: CtaVisSymbols.ImagePool.home_solo_black
        OnMouseClick: execute { ITF_DESCTOP_IN.HOME(); }
END_VISUALIZATION

// 40 Visualizations/DESCTOP/VIS_DESCTOP_APP_LINE
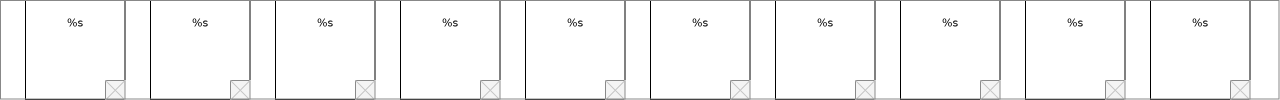
VISUALIZATION VIS_DESCTOP_APP_LINE  // 1280x100
VAR_INPUT
	usiStartNr		:	UsINT;
	ITF_DESCTOP_IN	:	ITF_DESCTOP;	
END_VAR
    Frame (25,0 100x100)
        shows VIS_APP(ITF_APP_IN := ITF_DESCTOP_IN.GET_APP(usiStartNr+ 0))
    Frame (150,0 100x100)
        shows VIS_APP(ITF_APP_IN := ITF_DESCTOP_IN.GET_APP(usiStartNr+ 1))
    Frame (275,0 100x100)
        shows VIS_APP(ITF_APP_IN := ITF_DESCTOP_IN.GET_APP(usiStartNr+ 2))
    Frame (400,0 100x100)
        shows VIS_APP(ITF_APP_IN := ITF_DESCTOP_IN.GET_APP(usiStartNr+ 3))
    Frame (525,0 100x100)
        shows VIS_APP(ITF_APP_IN := ITF_DESCTOP_IN.GET_APP(usiStartNr+ 4))
    Frame (650,0 100x100)
        shows VIS_APP(ITF_APP_IN := ITF_DESCTOP_IN.GET_APP(usiStartNr+ 5))
    Frame (775,0 100x100)
        shows VIS_APP(ITF_APP_IN := ITF_DESCTOP_IN.GET_APP(usiStartNr+ 6))
    Frame (900,0 100x100)
        shows VIS_APP(ITF_APP_IN := ITF_DESCTOP_IN.GET_APP(usiStartNr+ 7))
    Frame (1025,0 100x100)
        shows VIS_APP(ITF_APP_IN := ITF_DESCTOP_IN.GET_APP(usiStartNr+ 8))
    Frame (1150,0 100x100)
        shows VIS_APP(ITF_APP_IN := ITF_DESCTOP_IN.GET_APP(usiStartNr+ 9))
END_VISUALIZATION

// 40 Visualizations/DESCTOP/VIS_DESCTOP
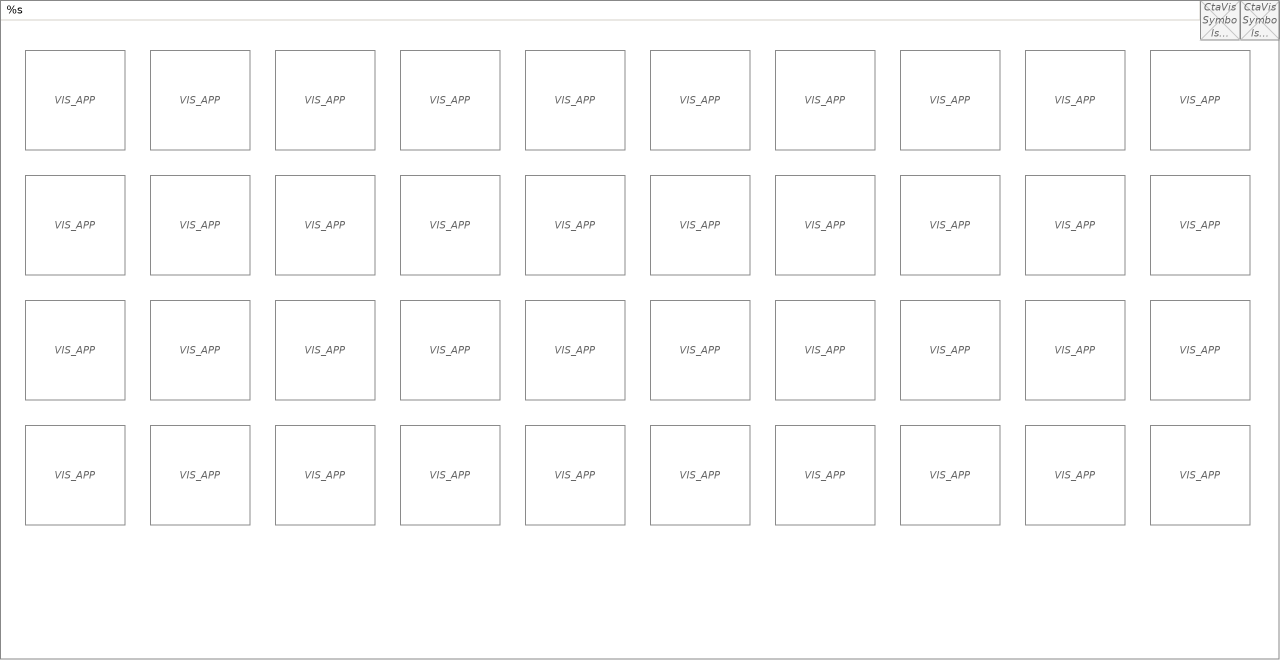
VISUALIZATION VIS_DESCTOP  // 1280x660
    Frame (0,0 1280x660)
        shows VIS_DESCTOP_GVL(ITF_DESCTOP_IN := GVL_VISU_APPS.DESCTOP)
END_VISUALIZATION
